FUNCTION_BLOCK FB_Receive
VAR_IN_OUT
	TxBuffer	: ComBuffer;
	RxBuffer	: ComBuffer;
END_VAR
VAR
	//Timer		: TON := (PT:=T#1S);
	//fbSend		: SendString;
	//bSendBusy	: BOOL;
	//eSendErrorID: ComError_t;
	//bReceivedByte	: BYTE;
	//bByteReceived	: BOOL;
	//bReceiveBusy	: BOOL;
	//bReceiveError	: BOOL;
	//bReceiveTimeout	: BOOL;
	fbReceive		: ReceiveByte;
	nReceiveCounter	: UDINT;
	bLastReceivedByte: BYTE;
	eReceiveErrorID	: ComError_t;
END_VAR

fbReceive(
//	Prefix:= '$02',
//	Suffix:= '$03',
//	Timeout:= T#1s,
//	ReceivedString:= bReceivedByte,
//	RxTimeout=> bReceiveTimeout 
//	ByteReceived=> bByteReceived,
//	Busy=> bReceiveBusy,
	RXbuffer:= RxBuffer,
	Error=> ,
	ByteReceived=>,
	ReceivedByte=>,
	);
IF fbReceive.Error <> COMERROR_NOERROR THEN
	eReceiveErrorID := fbReceive.Error;
END_IF
IF fbReceive.ByteReceived THEN
	nReceiveCounter := nReceiveCounter + 1;
	bLastReceivedByte := fbReceive.ReceivedByte;
END_IF

END_FUNCTION_BLOCK

(* stored: Version 1.1.0.1, ProductVersion 3.1.4024.11
   POU FB_Receive: Id {af516fa6-dd76-431e-80af-a81ebd3aa034}, SpecialFunc None *)
